PROGRAM Main
VAR
  ot : CL_LinkDefectMgrToTelegramAndLog;
END_VAR

ot();

END_PROGRAM

(* stored: Version 1.1.0.1, ProductVersion 3.1.4024.12
   POU Main: Id {3b58b2d0-00e0-4f0c-9117-84390552b287}, SpecialFunc None *)
